INTERFACE I_PersistentEventStorage

METHOD StoreEvent
VAR_INPUT
	stEvent : ST_Event;
END_VAR
END_METHOD

END_INTERFACE

(* stored: Version 1.1.0.1, ProductVersion 3.1.4024.10
   Itf I_PersistentEventStorage: Id {7e6adfce-a270-40e6-a471-4cc760d5b3a2}
   Method StoreEvent: Id {60a2d4a8-4400-406e-9230-6c0828dfd52d} *)
